(* Logix 5000 project; controller DispersionPlc vendor 1 type 14 code 108 rev 34.11; software revision 34.01; part 16 of 22 *)
(* tags used below, declared in another part *)
   _Placeholder_LS_4302_AI : REAL;
   AG4302_LLP_Alarm : BOOL;
   AG4302_LLPower : TIMER;
   Dummy_Safety_1 : BOOL[32];
   Estop_Disp : ALIAS FOR Local:3:I.Data.1;
   Fault_Reset_High : REAL;
   Faut_Reset_Low : REAL;
   FC_4302_1 : AStd_PIDInterface;
   FCV_4302_1 : AStd_VlvModulating;
   FCV_4302_1_AOI : AStd_VlVModulating_AOI;
   FE_4303_OffSet : REAL;
   FIT_4302_1 : AStd_AnalogInput;
   FIT_4302_1_AOI : AStd_AI_AOI;
   FIT_4302_1_Holding : DINT;
   FIT_4302_2 : AStd_AnalogInput;
   FIT_4302_2_AOI : AStd_AI_AOI;
   FIT_4302_2_Holding : DINT;
   FIT_4302_2_Samples : DINT;
   FLH : REAL;
   FLL : REAL;
   FQIC_4302_11_AOI : Analog_Scale;
   FQIC_4302_11_Corrected : REAL;
   FQIC_4302_11_Correction_Sf : REAL;
   FQIC_4302_11_Flow_Raw : DINT;
   FQIC_4302_11_OffSet_Out : REAL;
   FQIC_4302_11_Out : REAL;
   LS_4302_Dry : DINT;
   LS_4302_Faulted : BOOL;
   LS_4302_H_Off_Timer : TIMER;
   LS_4302_H_Timer : TIMER;
   LS_4302_High : BOOL;
   LS_4302_Wet : REAL;
   PCV_4302_3 : AStd_VlvModulating;
   PCV_4302_3_AOI : AStd_VlVModulating_AOI;
   PIC_4302_3 : AStd_PIDInterface;
   PIT_4302_2 : AStd_AnalogInput;
   PIT_4302_2_AOI : AStd_AI_AOI;
   PIT_4302_2_Holding : DINT;
   PIT_4302_2_Samples : DINT;
   PowerLimit : REAL;
   RO_HE4305_PhaseROHotWaterDrop : AStd_PLI;
   SPARE_O502 : ALIAS FOR Local:5:O.Data.2;
   SV_4302_1 : AStd_VlvOC;
   SV_4302_1_AOI : AStd_VlvOC_AOI;
   SV_4302_1_ICls : BOOL;
   SV_4302_1_OClose : BOOL;
   T4302_PhaseTempControl : AStd_PLI;
   TCV_4302_1 : AStd_VlvModulating;
   TCV_4302_1_AOI : AStd_VlVModulating_AOI;
   TCV_4302_2 : AStd_VlvModulating;
   TCV_4302_2_AOI : AStd_VlVModulating_AOI;
   TE_4302A : ALIAS FOR Local:8:I.Ch5Data;
   TIC_4302_4C : AStd_PIDInterface;
   TIC_4302_4H : AStd_PIDInterface;
   TIT_4302_1 : AStd_AnalogInput;
   TIT_4302_1_AOI : AStd_AI_AOI;
   TIT_4302_4 : AStd_AnalogInput;
   TIT_4302_4_AOI : AStd_AI_AOI;
   TIT_4302_5 : AStd_AnalogInput;
   TIT_4302_5_AOI : AStd_AI_AOI;
   VFD_4302_1 : AStd_VFD;
   VFD_4302_1_AOI : AStd_VFD_AOI;
   VFD_P_4302_2 : AStd_VFD;
   VFD_P_4302_2_AOI : AStd_VFD_AOI;
   XV_4302_10 : AStd_VlvOC;
(* Unit_S51, continued *)

ROUTINE MainRoutine   (* ladder *)
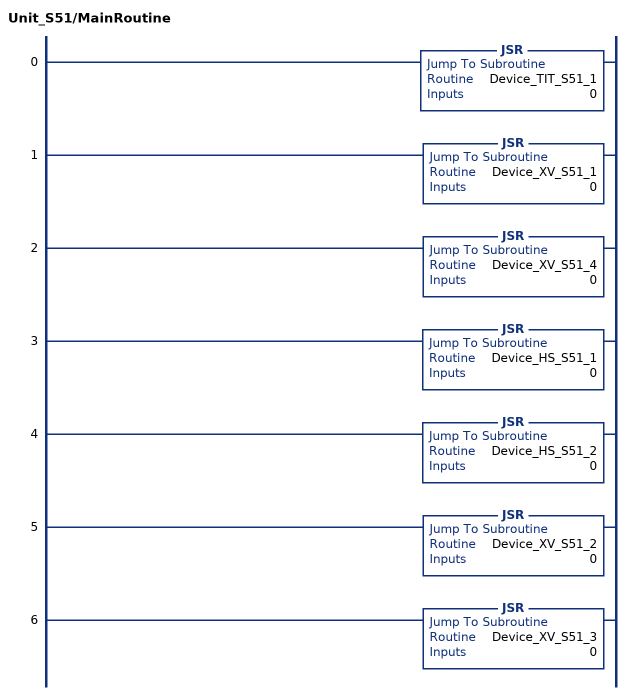
   0: JSR(Device_TIT_S51_1,0);
   1: JSR(Device_XV_S51_1,0);
   2: JSR(Device_XV_S51_4,0);
   3: JSR(Device_HS_S51_1,0);
   4: JSR(Device_HS_S51_2,0);
   5: JSR(Device_XV_S51_2,0);
   6: JSR(Device_XV_S51_3,0);
END_ROUTINE
END_PROGRAM

PROGRAM Unit_T4302   (* main routine MainRoutine *)

ROUTINE Device_FCV_4302_1   (* ladder *)
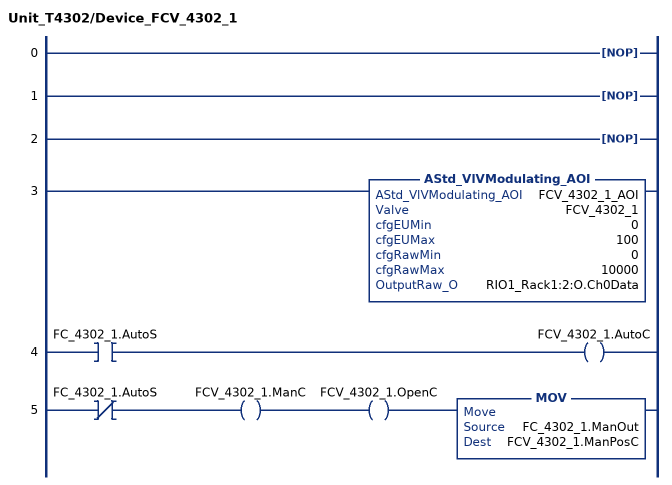
   0: NOP();
   1: NOP();
   2: NOP();
   3: AStd_VlVModulating_AOI(FCV_4302_1_AOI,FCV_4302_1,0,100,0,10000,RIO1_Rack1:2:O.Ch0Data);
   4: XIC(FC_4302_1.AutoS)OTE(FCV_4302_1.AutoC);
   5: XIO(FC_4302_1.AutoS)OTE(FCV_4302_1.ManC)OTE(FCV_4302_1.OpenC)MOV(FC_4302_1.ManOut,FCV_4302_1.ManPosC);
END_ROUTINE

ROUTINE Device_FIT_4302_1   (* ladder *)
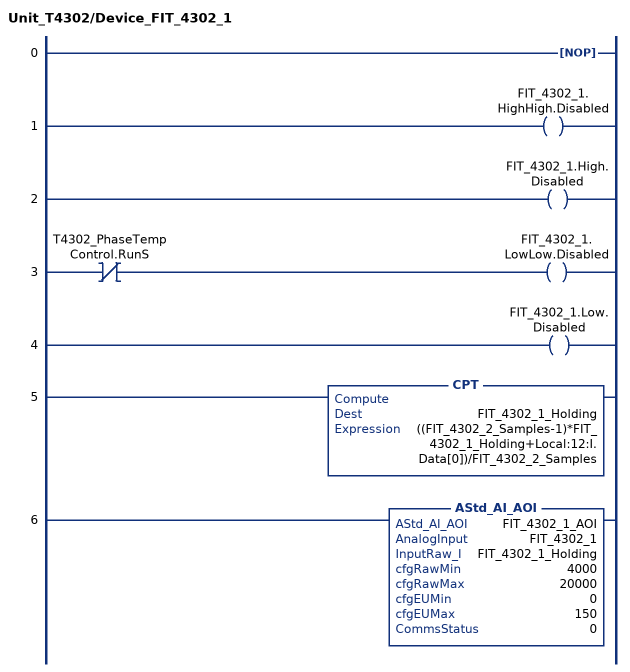
   0: NOP();
   1: OTE(FIT_4302_1.HighHigh.Disabled);
   2: OTE(FIT_4302_1.High.Disabled);
   3: XIO(T4302_PhaseTempControl.RunS)OTE(FIT_4302_1.LowLow.Disabled);
   4: OTE(FIT_4302_1.Low.Disabled);
   5: CPT(FIT_4302_1_Holding,((FIT_4302_2_Samples-1)*FIT_4302_1_Holding+Local:12:I.Data[0])/FIT_4302_2_Samples);
   6: AStd_AI_AOI(FIT_4302_1_AOI,FIT_4302_1,FIT_4302_1_Holding,4000,20000,0,150,0);
END_ROUTINE

ROUTINE Device_FIT_4302_2   (* ladder *)
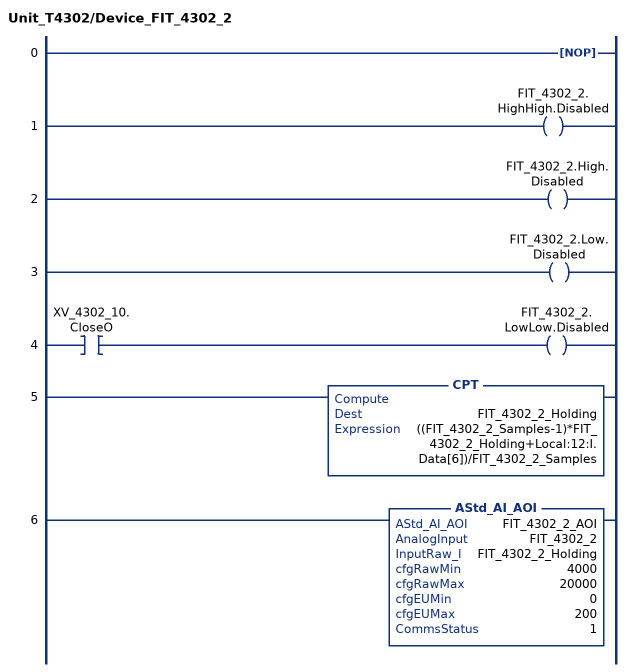
   0: NOP();
   1: OTE(FIT_4302_2.HighHigh.Disabled);
   2: OTE(FIT_4302_2.High.Disabled);
   3: OTE(FIT_4302_2.Low.Disabled);
   4: XIC(XV_4302_10.CloseO)OTE(FIT_4302_2.LowLow.Disabled);
   5: CPT(FIT_4302_2_Holding,((FIT_4302_2_Samples-1)*FIT_4302_2_Holding+Local:12:I.Data[6])/FIT_4302_2_Samples);
   6: AStd_AI_AOI(FIT_4302_2_AOI,FIT_4302_2,FIT_4302_2_Holding,4000,20000,0,200,1);
END_ROUTINE

ROUTINE Device_FQIC_4302_11   (* ladder *)
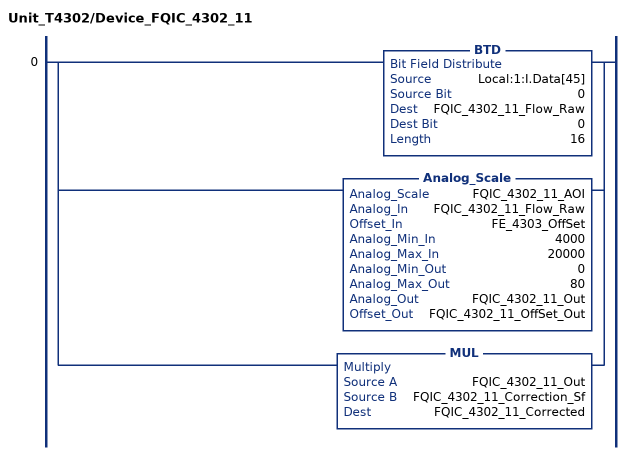
   0: [BTD(Local:1:I.Data[45],0,FQIC_4302_11_Flow_Raw,0,16) ,Analog_Scale(FQIC_4302_11_AOI,FQIC_4302_11_Flow_Raw,FE_4303_OffSet,4000,20000,0,80,FQIC_4302_11_Out,FQIC_4302_11_OffSet_Out) ,MUL(FQIC_4302_11_Out,FQIC_4302_11_Correction_Sf,FQIC_4302_11_Corrected) ];
END_ROUTINE

ROUTINE Device_LS_4302   (* ladder *)
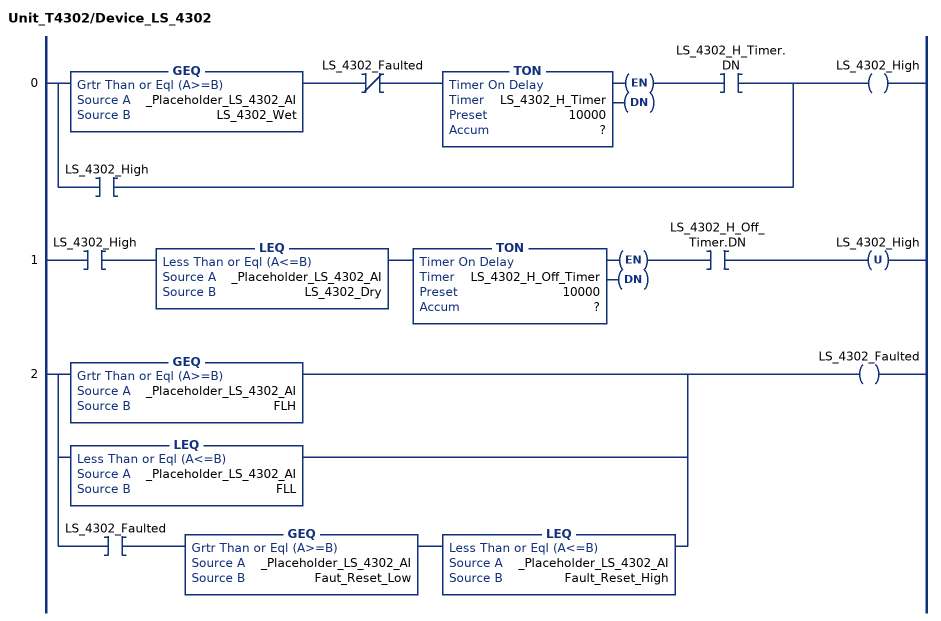
   0: [GEQ(_Placeholder_LS_4302_AI,LS_4302_Wet) XIO(LS_4302_Faulted) TON(LS_4302_H_Timer,?,?) XIC(LS_4302_H_Timer.DN) ,XIC(LS_4302_High) ]OTE(LS_4302_High);
   1: XIC(LS_4302_High)LEQ(_Placeholder_LS_4302_AI,LS_4302_Dry)TON(LS_4302_H_Off_Timer,?,?)XIC(LS_4302_H_Off_Timer.DN)OTU(LS_4302_High);
   2: [GEQ(_Placeholder_LS_4302_AI,FLH) ,LEQ(_Placeholder_LS_4302_AI,FLL) ,XIC(LS_4302_Faulted) GEQ(_Placeholder_LS_4302_AI,Faut_Reset_Low) LEQ(_Placeholder_LS_4302_AI,Fault_Reset_High) ]OTE(LS_4302_Faulted);
END_ROUTINE

ROUTINE Device_PCV_4302_3   (* ladder *)
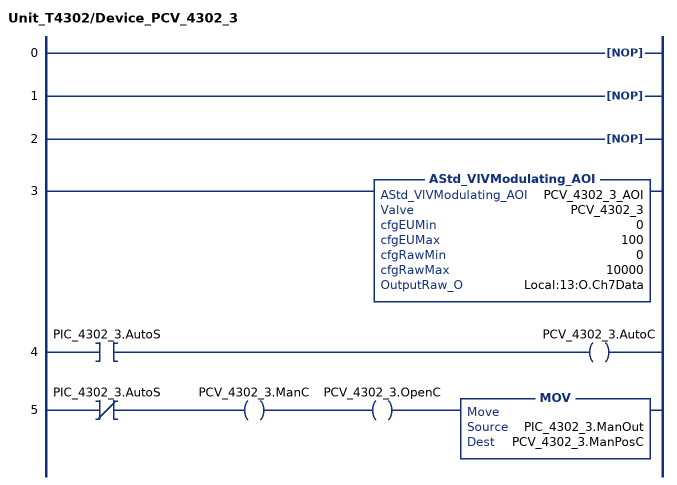
   0: NOP();
   1: NOP();
   2: NOP();
   3: AStd_VlVModulating_AOI(PCV_4302_3_AOI,PCV_4302_3,0,100,0,10000,Local:13:O.Ch7Data);
   4: XIC(PIC_4302_3.AutoS)OTE(PCV_4302_3.AutoC);
   5: XIO(PIC_4302_3.AutoS)OTE(PCV_4302_3.ManC)OTE(PCV_4302_3.OpenC)MOV(PIC_4302_3.ManOut,PCV_4302_3.ManPosC);
END_ROUTINE

ROUTINE Device_PIT_4302_2   (* ladder *)
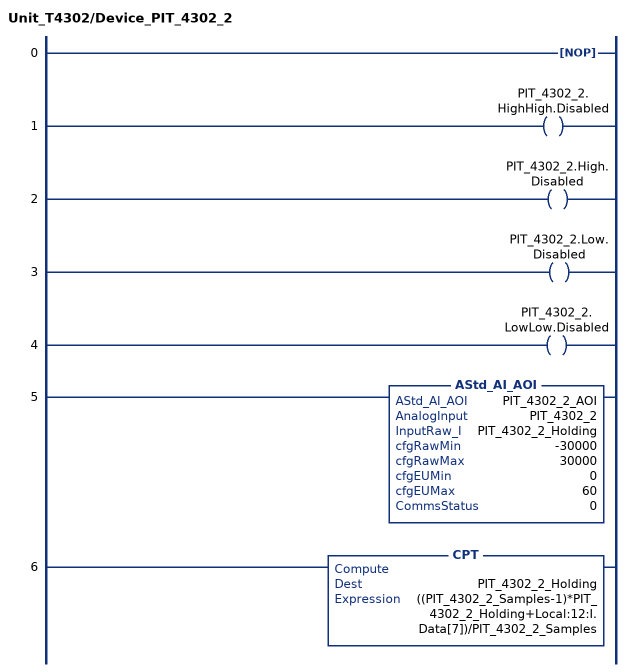
   0: NOP();
   1: OTE(PIT_4302_2.HighHigh.Disabled);
   2: OTE(PIT_4302_2.High.Disabled);
   3: OTE(PIT_4302_2.Low.Disabled);
   4: OTE(PIT_4302_2.LowLow.Disabled);
   5: AStd_AI_AOI(PIT_4302_2_AOI,PIT_4302_2,PIT_4302_2_Holding,-30000,30000,0,60,0);
   6: CPT(PIT_4302_2_Holding,((PIT_4302_2_Samples-1)*PIT_4302_2_Holding+Local:12:I.Data[7])/PIT_4302_2_Samples);
END_ROUTINE

ROUTINE Device_SV_4302_1   (* ladder *)
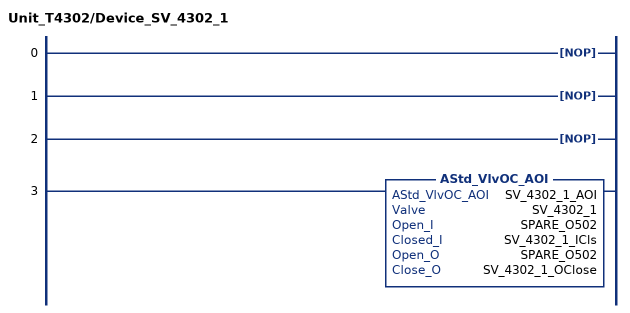
   0: NOP();
   1: NOP();
   2: NOP();
   3: AStd_VlvOC_AOI(SV_4302_1_AOI,SV_4302_1,SPARE_O502,SV_4302_1_ICls,SPARE_O502,SV_4302_1_OClose);
END_ROUTINE

ROUTINE Device_TCV_4302_1   (* ladder *)
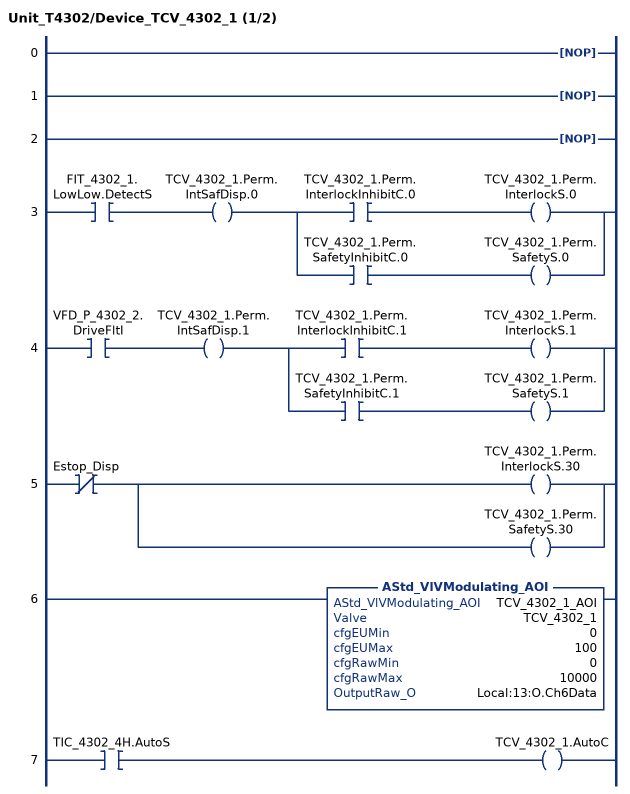
   0: NOP();
   1: NOP();
   2: NOP();
   3: XIC(FIT_4302_1.LowLow.DetectS)OTE(TCV_4302_1.Perm.IntSafDisp.0)[XIC(TCV_4302_1.Perm.InterlockInhibitC.0) OTE(TCV_4302_1.Perm.InterlockS.0) ,XIC(TCV_4302_1.Perm.SafetyInhibitC.0) OTE(TCV_4302_1.Perm.SafetyS.0) ];
   4: XIC(VFD_P_4302_2.DriveFltI)OTE(TCV_4302_1.Perm.IntSafDisp.1)[XIC(TCV_4302_1.Perm.InterlockInhibitC.1) OTE(TCV_4302_1.Perm.InterlockS.1) ,XIC(TCV_4302_1.Perm.SafetyInhibitC.1) OTE(TCV_4302_1.Perm.SafetyS.1) ];
   5: XIO(Estop_Disp)[OTE(TCV_4302_1.Perm.InterlockS.30) ,OTE(TCV_4302_1.Perm.SafetyS.30) ];
   6: AStd_VlVModulating_AOI(TCV_4302_1_AOI,TCV_4302_1,0,100,0,10000,Local:13:O.Ch6Data);
   7: XIC(TIC_4302_4H.AutoS)OTE(TCV_4302_1.AutoC);
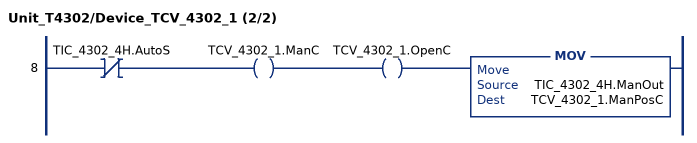
   8: XIO(TIC_4302_4H.AutoS)OTE(TCV_4302_1.ManC)OTE(TCV_4302_1.OpenC)MOV(TIC_4302_4H.ManOut,TCV_4302_1.ManPosC);
END_ROUTINE

ROUTINE Device_TCV_4302_2   (* ladder *)
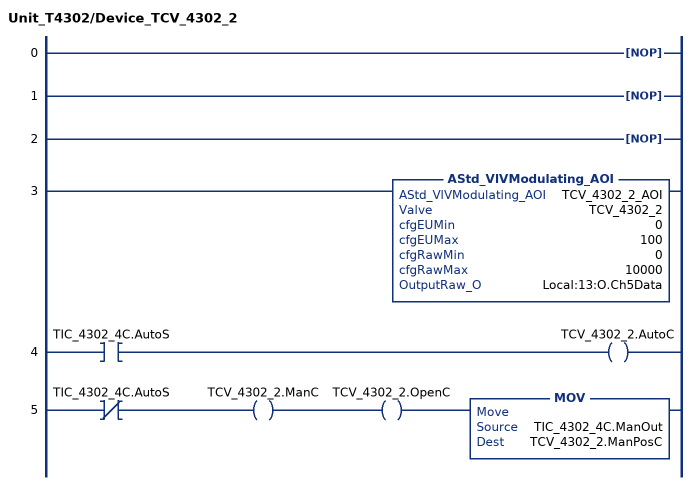
   0: NOP();
   1: NOP();
   2: NOP();
   3: AStd_VlVModulating_AOI(TCV_4302_2_AOI,TCV_4302_2,0,100,0,10000,Local:13:O.Ch5Data);
   4: XIC(TIC_4302_4C.AutoS)OTE(TCV_4302_2.AutoC);
   5: XIO(TIC_4302_4C.AutoS)OTE(TCV_4302_2.ManC)OTE(TCV_4302_2.OpenC)MOV(TIC_4302_4C.ManOut,TCV_4302_2.ManPosC);
END_ROUTINE

ROUTINE Device_TIT_4302_1   (* ladder *)
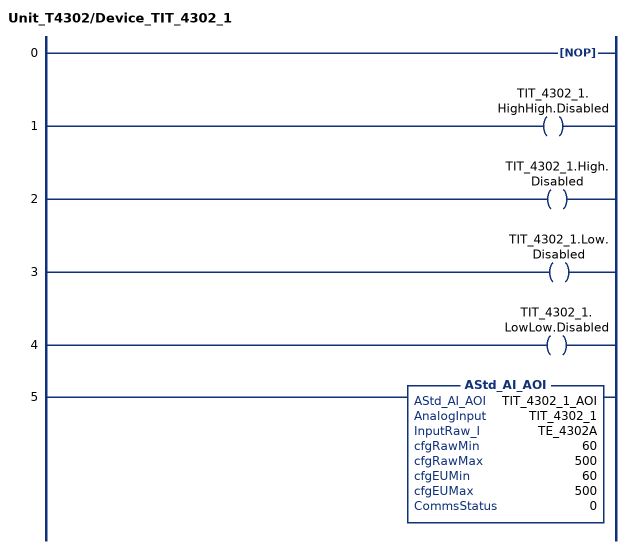
   0: NOP();
   1: OTE(TIT_4302_1.HighHigh.Disabled);
   2: OTE(TIT_4302_1.High.Disabled);
   3: OTE(TIT_4302_1.Low.Disabled);
   4: OTE(TIT_4302_1.LowLow.Disabled);
   5: AStd_AI_AOI(TIT_4302_1_AOI,TIT_4302_1,TE_4302A,60,500,60,500,0);
END_ROUTINE

ROUTINE Device_TIT_4302_4   (* ladder *)
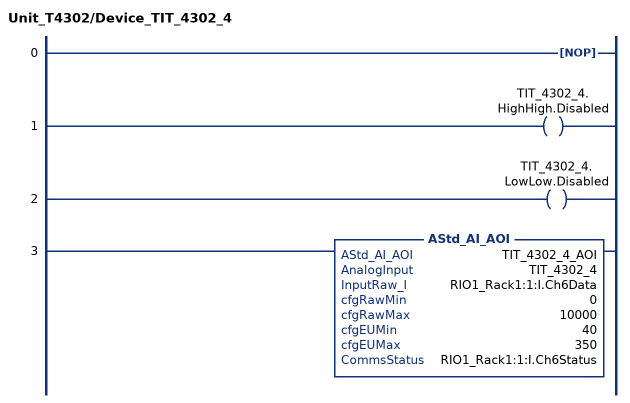
   0: NOP();
   1: OTE(TIT_4302_4.HighHigh.Disabled);
   2: OTE(TIT_4302_4.LowLow.Disabled);
   3: AStd_AI_AOI(TIT_4302_4_AOI,TIT_4302_4,RIO1_Rack1:1:I.Ch6Data,0,10000,40,350,RIO1_Rack1:1:I.Ch6Status);
END_ROUTINE

ROUTINE Device_TIT_4302_5   (* ladder *)
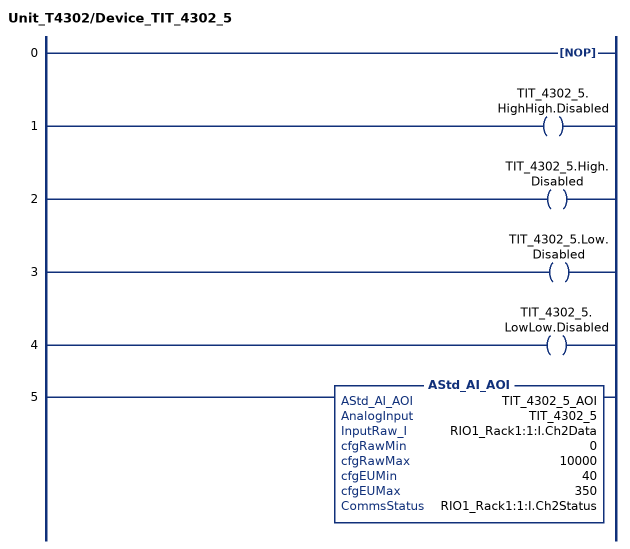
   0: NOP();
   1: OTE(TIT_4302_5.HighHigh.Disabled);
   2: OTE(TIT_4302_5.High.Disabled);
   3: OTE(TIT_4302_5.Low.Disabled);
   4: OTE(TIT_4302_5.LowLow.Disabled);
   5: AStd_AI_AOI(TIT_4302_5_AOI,TIT_4302_5,RIO1_Rack1:1:I.Ch2Data,0,10000,40,350,RIO1_Rack1:1:I.Ch2Status);
END_ROUTINE

ROUTINE Device_VFD_4302_1   (* ladder *)
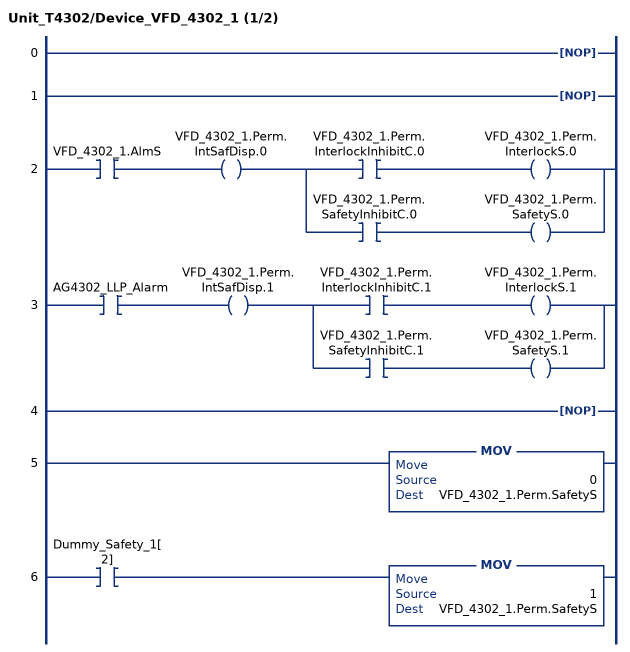
   0: NOP();
   1: NOP();
   2: XIC(VFD_4302_1.AlmS)OTE(VFD_4302_1.Perm.IntSafDisp.0)[XIC(VFD_4302_1.Perm.InterlockInhibitC.0) OTE(VFD_4302_1.Perm.InterlockS.0) ,XIC(VFD_4302_1.Perm.SafetyInhibitC.0) OTE(VFD_4302_1.Perm.SafetyS.0) ];
   3: XIC(AG4302_LLP_Alarm)OTE(VFD_4302_1.Perm.IntSafDisp.1)[XIC(VFD_4302_1.Perm.InterlockInhibitC.1) OTE(VFD_4302_1.Perm.InterlockS.1) ,XIC(VFD_4302_1.Perm.SafetyInhibitC.1) OTE(VFD_4302_1.Perm.SafetyS.1) ];
   4: NOP();
   5: MOV(0,VFD_4302_1.Perm.SafetyS);
   6: XIC(Dummy_Safety_1[2])MOV(1,VFD_4302_1.Perm.SafetyS);
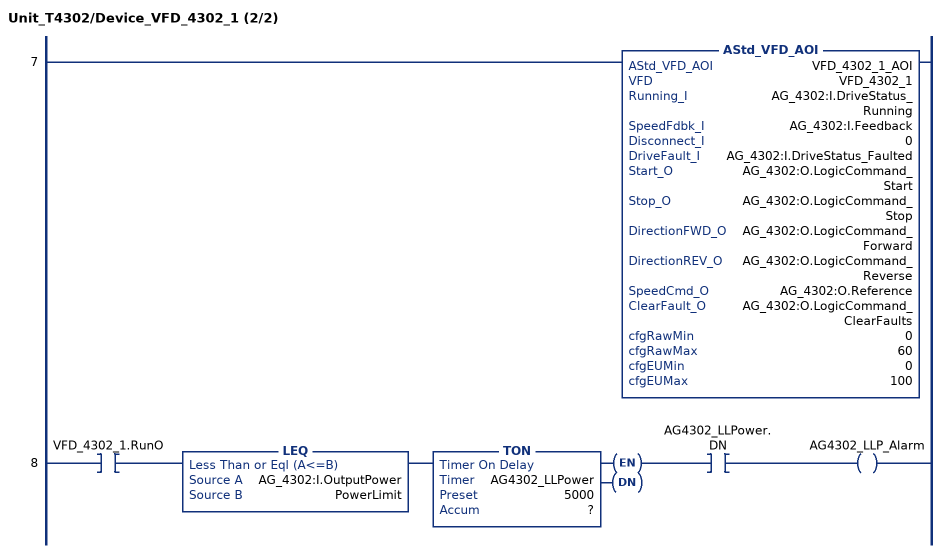
   7: AStd_VFD_AOI(VFD_4302_1_AOI,VFD_4302_1,AG_4302:I.DriveStatus_Running,AG_4302:I.Feedback,0,AG_4302:I.DriveStatus_Faulted,AG_4302:O.LogicCommand_Start,AG_4302:O.LogicCommand_Stop,AG_4302:O.LogicCommand_Forward,AG_4302:O.LogicCommand_Reverse,AG_4302:O.Reference,AG_4302:O.LogicCommand_ClearFaults,0,60,0,100);
   8: XIC(VFD_4302_1.RunO)LEQ(AG_4302:I.OutputPower,PowerLimit)TON(AG4302_LLPower,?,?)XIC(AG4302_LLPower.DN)OTE(AG4302_LLP_Alarm);
END_ROUTINE

ROUTINE Device_VFD_P_4302_2   (* ladder *)
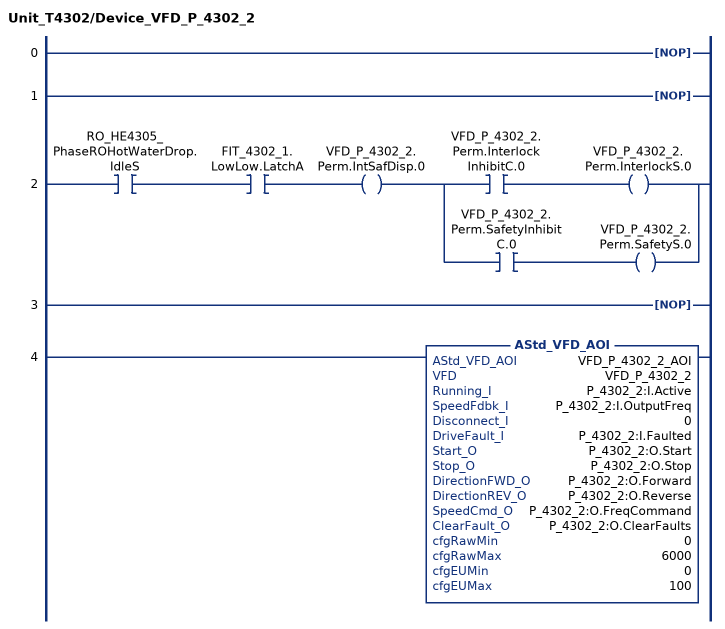
   0: NOP();
   1: NOP();
   2: XIC(RO_HE4305_PhaseROHotWaterDrop.IdleS)XIC(FIT_4302_1.LowLow.LatchA)OTE(VFD_P_4302_2.Perm.IntSafDisp.0)[XIC(VFD_P_4302_2.Perm.InterlockInhibitC.0) OTE(VFD_P_4302_2.Perm.InterlockS.0) ,XIC(VFD_P_4302_2.Perm.SafetyInhibitC.0) OTE(VFD_P_4302_2.Perm.SafetyS.0) ];
   3: NOP();
   4: AStd_VFD_AOI(VFD_P_4302_2_AOI,VFD_P_4302_2,P_4302_2:I.Active,P_4302_2:I.OutputFreq,0,P_4302_2:I.Faulted,P_4302_2:O.Start,P_4302_2:O.Stop,P_4302_2:O.Forward,P_4302_2:O.Reverse,P_4302_2:O.FreqCommand,P_4302_2:O.ClearFaults,0,6000,0,100);
END_ROUTINE
